FUNCTION_BLOCK FB_BoxLED
VAR_INPUT
END_VAR
VAR_OUTPUT
	eCondition : eConditionCheck;
END_VAR
VAR
	eLEDMode : eLightMode;
END_VAR

PROPERTY setLightMode : eLightMode
SET
eLEDMode := setLightMode;
END_SET
END_PROPERTY

END_FUNCTION_BLOCK

(* stored: Version 1.1.0.1, ProductVersion 3.1.4024.12
   POU FB_BoxLED: Id {55242ab5-9ff4-4666-b1b6-38e99286d969}, SpecialFunc None
   Property setLightMode: Id {8039be3d-e687-4f0b-a7ec-3b99ee8a857e}
   Set Set: Id {ab54af1d-7396-4390-94b5-279c607d86d7} *)
